(* IEC 61131-3 sources: CodesysTest/export/Pro24.dev/Plc Logic/Application/Pro24/Applied Motion/FB_AppliedMotionStepServoEIPBaseQX.pou/Faulted.prop, 1 file *)

(* ---- Get.pm.st ---- *)
(*#-#-#-#-#-#-#-#-#-#---Declaration---#-#-#-#-#-#-#-#-#-#-#-#-#*)

VAR
END_VAR
(*#-#-#-#-#-#-#-#-#-#---Implementation---#-#-#-#-#-#-#-#-#-#-#-#-#*)

Faulted := _faulted;
